Staubli VAL3: EnterPageKey.pgx

program EnterPageKey(num& x_nKey (dimensions=1), num& x_nSelect (dimensions=1), string& x_sItem (dimensions=1), trsf& x_trOffset (dimensions=1))
  local bool l_bRes
  local num l_nItem
  local num l_nKey
  local num l_nView
  local string l_sItem
  local string l_sStr
  local string l_sValue
  local string l_sYN[2]
  local point lp
begin
  //
  if x_nKey==270
    switch x_nSelect
      case 0

        call user:editNum(x_sItem,sListItemValue[x_nSelect],x_trOffset.x,x_nSelect)

      break
      //
      case 1

        call user:editNum(x_sItem,sListItemValue[x_nSelect],x_trOffset.y,x_nSelect)

      break
      //
      case 2

        call user:editNum(x_sItem,sListItemValue[x_nSelect],x_trOffset.z,x_nSelect)

      break
    endSwitch
    bUserRefresh=true
    bListRefresh=true
  endIf
end
